Staubli VAL3: getInstr.pgx

public program getInstr(InstrItem& x_iInstr[], bool x_bType, num x_nIndex)
  local string l_sInstruction
  local num i
begin
  // get the instruction and fill as an array
  if x_nIndex>=0
    if x_bType
      // take gun ON
      //resize(x_iInstr,1,size(saveData:tData[x_nIndex].iActionON))
      for i=0 to size(x_iInstr)-1
        x_iInstr[i]=saveData:tData[x_nIndex].iActionON[i]
      endFor
    else
      // take gun OFF
      //resize(x_iInstr,1,size(saveData:tData[x_nIndex].iActionOFF))
      for i=0 to size(x_iInstr)-1
        x_iInstr[i]=saveData:tData[x_nIndex].iActionOFF[i]
      endFor
    endIf
  endIf
end
